(*
	Return the low byte from the input word
*)
FUNCTION F_GetLByte : BYTE
VAR_INPUT
	nWord	: WORD;
END_VAR

F_GetLByte := WORD_TO_BYTE(nWord);

END_FUNCTION

(* stored: Version 1.1.0.1, ProductVersion 3.1.4024.12
   POU F_GetLByte: Id {cd10e641-289c-00b7-336d-c4f34a4bdec1}, SpecialFunc None *)
